// TIA Portal V20 export
VAR_GLOBAL   // PLC tag table "LKinCtrl_HMI_Editor_Messages"
END_VAR
VAR_GLOBAL CONSTANT   // user constants
   LKINCTRL_MESSAGEID_POINT_DELETE : Int := 101;   // Info: 1-6999, Warning: 7000-7999, Error: 8000-
   LKINCTRL_MESSAGEID_COPY : Int := 1;   // Info: 1-6999, Warning: 7000-7999, Error: 8000-
   LKINCTRL_MESSAGEID_REDO : Int := 21;   // Info: 1-6999, Warning: 7000-7999, Error: 8000-
   LKINCTRL_MESSAGEID_MULTI_ON : Int := 10;   // Info: 1-6999, Warning: 7000-7999, Error: 8000-
   LKINCTRL_MESSAGEID_PASTE : Int := 2;   // Info: 1-6999, Warning: 7000-7999, Error: 8000-
   LKINCTRL_MESSAGEID_MULTI_OFF : Int := 11;   // Info: 1-6999, Warning: 7000-7999, Error: 8000-
   LKINCTRL_MESSAGEID_POINT_SAVE : Int := 100;   // Info: 1-6999, Warning: 7000-7999, Error: 8000-
   LKINCTRL_MESSAGEID_UNDO : Int := 20;   // Info: 1-6999, Warning: 7000-7999, Error: 8000-
   LKINCTRL_MESSAGEID_ADD_NEW : Int := 3;   // Info: 1-6999, Warning: 7000-7999, Error: 8000-
   LKINCTRL_MESSAGEID_DELETE : Int := 4;   // Info: 1-6999, Warning: 7000-7999, Error: 8000-
   LKINCTRL_MESSAGEID_PATH_FULL : Int := 8001;   // Info: 1-6999, Warning: 7000-7999, Error: 8000-
   LKINCTRL_MESSAGEID_NO_AUX_POINT : Int := 8000;   // Info: 1-6999, Warning: 7000-7999, Error: 8000-
   LKINCTRL_MESSAGEID_POINT_CONVERT : Int := 102;   // Info: 1-6999, Warning: 7000-7999, Error: 8000-
   LKINCTRL_MESSAGEID_POINT_UNDO : Int := 103;   // Info: 1-6999, Warning: 7000-7999, Error: 8000-
   LKINCTRL_MESSAGEID_POINT_REDO : Int := 104;   // Info: 1-6999, Warning: 7000-7999, Error: 8000-
   LKINCTRL_MESSAGEID_POINT_LINKCONST_COPIED : Int := 107;   // Info: 1-6999, Warning: 7000-7999, Error: 8000-
   LKINCTRL_MESSAGEID_POINT_TJ_COPIED : Int := 106;   // Info: 1-6999, Warning: 7000-7999, Error: 8000-
   LKINCTRL_MESSAGEID_POINT_POSITION_COPIED : Int := 105;   // Info: 1-6999, Warning: 7000-7999, Error: 8000-
   LKINCTRL_MESSAGEID_POINT_POSE_COPIED : Int := 108;   // Info: 1-6999, Warning: 7000-7999, Error: 8000-
   LKINCTRL_MESSAGEID_POINT_TOUCHUP : Int := 109;   // Info: 1-6999, Warning: 7000-7999, Error: 8000-
   LKINCTRL_MESSAGEID_TOUCHUP : Int := 5;   // Info: 1-6999, Warning: 7000-7999, Error: 8000-
END_VAR
